{attribute 'OPC.UA.DA' := '1'}
{attribute 'OPC.UA.DA.StructuredType' := '1'}
TYPE ResponsivityMsg :
STRUCT
	Id : EPowerIlluminationFlow;
	Responsivity : LREAL;
END_STRUCT
END_TYPE

(* stored: Version 1.1.0.1, ProductVersion 3.1.4024.10
   DUT ResponsivityMsg: Id {88c831cc-b3fe-4953-baf4-618a49623485} *)
